Fanuc KAREL source: kt00415.KL

-- PROVISIONAL review KL for V940-1; original PC SHA256 ccac4e3a1551f506f138b3df08db635002eb2a9d77893b699c07d3a47231c81f
-- Incomplete behavior may be omitted. Consult companion uncertainty JSON. Do not deploy.
PROGRAM KT00415
%NOLOCKGROUP
VAR
  I2 : INTEGER
  OUT : BOOLEAN
-- UNRESOLVED_DECL H1 type=002017
BEGIN
  -- V9_ZERO_TABLE_METADATA_HINT layout=0001; no indexed target words; source/name/runtime held
  -- UNRESOLVED_PC offsets 5-19; opcodes 2E,22,9D,33,B4
  -- UNRESOLVED_PC offsets 24-35; opcodes 2E,23
  -- UNRESOLVED_PC offsets 40-62; opcodes 22,9D,33,B3,21,5B,23
  -- UNRESOLVED_PC offsets 67-71; opcodes 7F
END KT00415
